Fanuc KAREL source: ko00033.KL

PROGRAM KO00033
%STACKSIZE=65535
%PRIORITY=65535
%NOLOCKGROUP
VAR
P1 : POSITION
P2 : POSITION
F : BOOLEAN
OUT : POSITION
BEGIN
F=TRUE
-- UNSAFE_SOURCE_IR line 11: CALL_RESULT MIRROR(convert_position_to_xyzwprext(P1), P2, F)
END KO00033
